VAR_GLOBAL
    (* Written by TestHarness or simulation environment. bSimulationMode must be TRUE. *)
    stVirtualIO : ST_VirtualIO;
END_VAR

(* stored: Version 1.1.0.1
   GVL GVL_VirtualIO: Id {806793BF-235B-3FE2-7581-BBD9E112F769} *)
